Yaskawa INFORM job: R1_W29-KM-NOWY.JBI

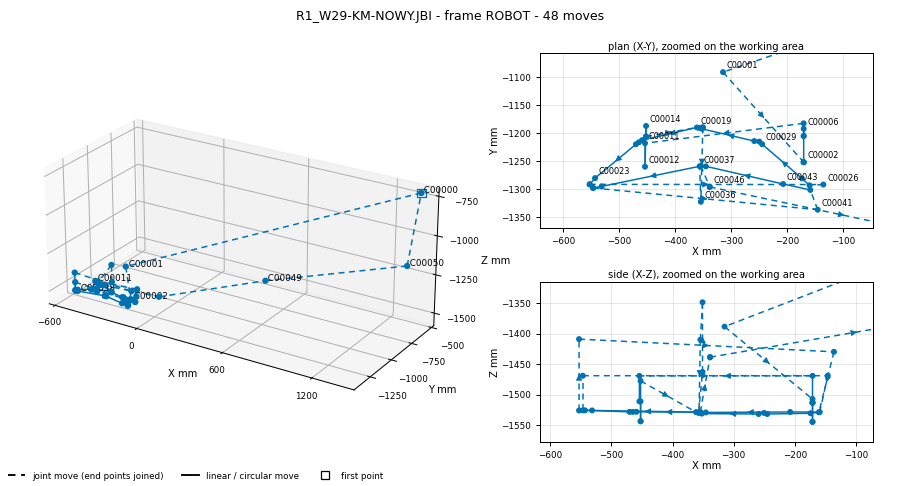
[picture p0: tool path of R1_W29-KM-NOWY.JBI in frame ROBOT, 48 of 48 moves have a stored position in this frame; points joined in program order, loops and branches not executed]
/JOB
//NAME R1_W29-KM-NOWY
///FOLDERNAME KRIS-SCIANA
//POS
///NPOS 52,52,48,3,0,0
///TOOL 0
///POSTYPE ROBOT
///RECTAN
///RCONF 0,0,0,0,0,0,0,0,0,0,0,0,0,0,0,0,0,0,0,0,0,0,0,0
C00000=1380.020,-512.213,-734.768,45.7984,-2.5734,-62.2106
C00001=-314.885,-1091.342,-1388.620,7.0991,47.6528,95.5247
C00002=-170.882,-1252.122,-1507.196,7.0965,47.6516,95.5184
C00003=-170.878,-1252.127,-1513.169,7.0965,47.6519,95.5192
C00004=-170.856,-1252.136,-1525.077,7.0962,47.6516,95.5223
C00005=-170.878,-1252.127,-1513.169,7.0965,47.6519,95.5192
C00006=-170.880,-1192.452,-1513.156,7.0958,47.6523,95.5184
C00007=-170.881,-1205.262,-1544.508,7.0940,47.6532,95.5150
C00008=-170.883,-1210.138,-1544.498,7.0940,47.6527,95.5159
C00009=-170.881,-1205.262,-1544.508,7.0940,47.6532,95.5150
C00010=-170.885,-1182.718,-1469.214,7.0949,47.6534,95.5162
C00011=-454.226,-1218.230,-1469.227,7.0938,47.6529,95.5164
C00012=-454.225,-1260.141,-1510.984,7.0936,47.6521,95.5169
C00013=-454.221,-1260.145,-1522.091,7.0917,47.6525,95.5139
C00014=-452.331,-1187.443,-1510.977,7.0932,47.6531,95.5154
C00015=-452.309,-1206.496,-1543.511,7.0905,47.6535,95.5128
C00016=-452.283,-1211.717,-1543.520,7.0889,47.6539,95.5119
C00017=-452.309,-1206.496,-1543.511,7.0905,47.6535,95.5128
C00018=-452.308,-1206.485,-1477.500,7.0906,47.6527,95.5130
C00019=-361.495,-1190.117,-1528.559,4.0105,46.8580,82.9369
C00020=-459.241,-1212.758,-1528.059,4.0090,46.8598,82.9290
C00021=-465.152,-1216.573,-1528.195,4.0138,46.8598,102.2526
C00022=-470.424,-1220.169,-1528.108,4.0135,46.8596,110.5818
C00023=-543.410,-1280.537,-1525.621,4.0159,46.8611,110.5850
C00024=-553.033,-1291.721,-1525.884,4.0182,46.8612,110.5866
C00025=-553.029,-1291.719,-1409.041,4.0170,46.8613,110.5846
C00026=-135.797,-1292.057,-1429.838,4.0180,46.8613,34.2800
C00027=-160.429,-1293.450,-1528.859,4.0112,46.8630,34.2695
C00028=-174.166,-1280.960,-1530.412,4.0163,46.8653,34.2766
C00029=-245.014,-1220.022,-1531.655,4.0137,46.8657,34.2760
C00030=-250.213,-1215.388,-1529.872,4.0121,46.8638,62.9323
C00031=-259.100,-1214.397,-1531.605,4.0118,46.8648,62.9324
C00032=-352.156,-1192.622,-1530.999,4.0138,46.8647,62.9360
C00033=-357.322,-1190.843,-1529.939,4.0131,46.8635,62.9345
C00034=-350.946,-1189.951,-1462.802,4.0124,46.8636,62.9333
C00035=-350.944,-1189.951,-1348.723,4.0127,46.8636,62.9343
C00036=-354.498,-1322.808,-1410.027,-15.4920,32.5646,-91.9565
C00037=-356.649,-1259.427,-1528.581,-15.4938,32.5644,-91.9586
C00038=-531.724,-1295.391,-1525.761,-15.4977,32.5637,-91.9664
C00039=-546.841,-1298.072,-1525.633,-15.4952,32.5617,-91.9642
C00040=-546.841,-1298.137,-1468.923,-15.4951,32.5627,-91.9631
C00041=-145.871,-1337.003,-1468.926,-15.4954,32.5637,-91.9623
C00042=-159.004,-1301.691,-1528.387,-15.4958,32.5640,-91.9617
C00043=-207.491,-1291.075,-1528.320,-15.4966,32.5644,-91.9616
C00044=-345.558,-1259.505,-1529.077,-15.4968,32.5617,-91.9666
C00045=-354.594,-1258.772,-1528.388,-15.4965,32.5625,-91.9640
C00046=-338.619,-1296.215,-1438.631,-18.1913,27.2183,-112.1098
C00047=-338.616,-1296.213,-1438.634,-18.1910,27.2179,-81.5660
C00048=133.748,-1396.204,-1357.645,-19.2328,23.1684,-62.3382
C00049=800.262,-1291.531,-1131.161,-1.6815,44.3835,75.7924
C00050=1382.830,-664.674,-1139.962,22.7477,31.6881,-179.3432
C00051=1380.020,-512.213,-734.768,45.7984,-2.5734,-62.2106
BC00000=786.429,2790.581,1999.643
BC00001=1673.587,2787.026,1999.675
BC00002=1673.587,2787.026,1999.675
BC00003=1673.587,2787.026,1999.675
BC00004=1673.587,2787.026,1999.675
BC00005=1673.587,2787.026,1999.675
BC00006=1673.587,2787.026,1999.675
BC00007=1673.587,2787.026,1999.675
BC00008=1673.587,2787.026,1999.675
BC00009=1673.587,2787.026,1999.675
BC00010=1673.587,2787.026,1999.675
BC00011=1673.587,2787.026,1999.675
BC00012=1673.587,2787.026,1999.675
BC00013=1673.587,2787.026,1999.675
BC00014=1673.587,2787.026,1999.675
BC00015=1673.587,2787.026,1999.675
BC00016=1673.587,2787.026,1999.675
BC00017=1673.587,2787.026,1999.675
BC00018=1673.587,2787.026,1999.675
BC00019=1724.246,2786.825,1999.677
BC00020=1724.246,2786.825,1999.677
BC00021=1724.246,2786.825,1999.677
BC00022=1724.246,2786.825,1999.677
BC00023=1724.246,2786.825,1999.677
BC00024=1724.246,2786.825,1999.677
BC00025=1724.246,2786.825,1999.677
BC00026=1724.246,2786.825,1999.677
BC00027=1724.246,2786.825,1999.677
BC00028=1724.246,2786.825,1999.677
BC00029=1724.246,2786.825,1999.677
BC00030=1724.246,2786.825,1999.677
BC00031=1724.246,2786.825,1999.677
BC00032=1724.246,2786.825,1999.677
BC00033=1724.246,2786.825,1999.677
BC00034=1724.246,2786.825,1999.677
BC00035=1724.246,2786.825,1999.677
BC00036=1724.246,2786.825,1999.677
BC00037=1724.246,2786.825,1999.677
BC00038=1724.246,2786.825,1999.677
BC00039=1724.246,2786.825,1999.677
BC00040=1724.246,2786.825,1999.677
BC00041=1724.246,2786.825,1999.677
BC00042=1724.246,2786.825,1999.677
BC00043=1724.246,2786.825,1999.677
BC00044=1724.246,2786.825,1999.677
BC00045=1724.246,2786.825,1999.677
BC00046=1724.246,2786.825,1999.677
BC00047=1724.246,2786.825,1999.677
BC00048=1442.256,2786.825,1999.677
BC00049=812.904,2786.825,1999.677
BC00050=213.733,2786.825,1999.677
BC00051=786.429,2790.581,1999.643
///POSTYPE PULSE
///PULSE
EC00000=798155,-556476
EC00001=798156,-556476
EC00002=798156,-556476
EC00003=798156,-556476
EC00004=798156,-556476
EC00005=798156,-556476
EC00006=798156,-556476
EC00007=798156,-556476
EC00008=798156,-556476
EC00009=798156,-556476
EC00010=798156,-556476
EC00011=798156,-556476
EC00012=798156,-556476
EC00013=798156,-556476
EC00014=798156,-556476
EC00015=798156,-556476
EC00016=798156,-556476
EC00017=798156,-556476
EC00018=798156,-556476
EC00019=798156,-556476
EC00020=798156,-556476
EC00021=798156,-556476
EC00022=798156,-556476
EC00023=798156,-556476
EC00024=798156,-556476
EC00025=798156,-556476
EC00026=798156,-556476
EC00027=798156,-556476
EC00028=798156,-556476
EC00029=798156,-556476
EC00030=798156,-556476
EC00031=798156,-556476
EC00032=798156,-556476
EC00033=798156,-556476
EC00034=798156,-556476
EC00035=798156,-556476
EC00036=798156,-556476
EC00037=798156,-556476
EC00038=798156,-556476
EC00039=798156,-556476
EC00040=798156,-556476
EC00041=798156,-556476
EC00042=798156,-556476
EC00043=798156,-556476
EC00044=798156,-556476
EC00045=798156,-556476
EC00046=798156,-556476
EC00047=798155,-556476
///POSTYPE BASE
///RECTAN
///RCONF 0,0,0,0,1,0,0,0,0,0,0,0,0,0,0,0,0,0,0,0,0,0,0,0
P00006=2.006,1.622,-0.565,0.0000,0.0000,0.0000
P00021=0.073,2.058,-0.109,0.0000,0.0000,0.0000
P00022=2.006,1.622,-0.565,0.0000,0.0000,0.0000
//INST
///DATE 2024/02/06 17:41
///ATTR SC,RW,RJ
////FRAME ROBOT
///GROUP1 RB1,BS1
///GROUP2 ST1
NOP
MOVJ C00000 BC00000 VJ=15.00  +MOVJ EC00000 VJ=15.00
MOVJ C00001 BC00001 VJ=50.00  +MOVJ EC00001 VJ=50.00
MOVJ C00002 BC00002 VJ=15.00  +MOVJ EC00002 VJ=15.00
MOVL C00003 BC00003 V=58.3  +MOVJ EC00003 VJ=15.00
REFP 3 RB1 C00004 BC00004
CALL JOB:SEARCH-R1
SET P021 P006
SFTON P021
MOVL C00005 BC00005 V=58.3  +MOVJ EC00004 VJ=15.00
MOVL C00006 BC00006 V=58.3  +MOVJ EC00005 VJ=15.00
MOVL C00007 BC00007 V=58.3  +MOVJ EC00006 VJ=15.00
REFP 3 RB1 C00008 BC00008
CALL JOB:SEARCH-R1
SET P021 P006
SFTON P021
MOVL C00009 BC00009 V=58.3  +MOVJ EC00007 VJ=15.00
SFTOF
MOVL C00010 BC00010 V=133.3  +MOVJ EC00008 VJ=15.00
MOVJ C00011 BC00011 VJ=15.00  +MOVJ EC00009 VJ=15.00
MOVL C00012 BC00012 V=58.3  +MOVJ EC00010 VJ=15.00
REFP 3 RB1 C00013 BC00013
CALL JOB:SEARCH-R1
SET P022 P006
SFTON P022
MOVL C00014 BC00014 V=58.3  +MOVJ EC00011 VJ=15.00
MOVL C00015 BC00015 V=58.3  +MOVJ EC00012 VJ=15.00
REFP 3 RB1 C00016 BC00016
CALL JOB:SEARCH-R1
SET P022 P006
SFTON P022
MOVL C00017 BC00017 V=58.3  +MOVJ EC00013 VJ=15.00
SFTOF
MOVL C00018 BC00018 V=133.3  +MOVJ EC00014 VJ=15.00
SFTON P022
MOVJ C00019 BC00019 VJ=15.00  +MOVJ EC00015 VJ=50.00
MACRO1 MJ#(0) ARGF7
ARCON
MOVL C00020 BC00020 V=10.8  +MOVJ EC00016 VJ=15.00
MOVL C00021 BC00021 V=10.8  +MOVJ EC00017 VJ=15.00
MOVL C00022 BC00022 V=10.8  +MOVJ EC00018 VJ=15.00
MOVL C00023 BC00023 V=10.8  +MOVJ EC00019 VJ=15.00
MOVL C00024 BC00024 V=10.8  +MOVJ EC00020 VJ=15.00
ARCOF
SFTOF
MOVJ C00025 BC00025 VJ=15.00  +MOVJ EC00021 VJ=15.00
MOVJ C00026 BC00026 VJ=15.00  +MOVJ EC00022 VJ=15.00
SFTON P021
MOVJ C00027 BC00027 VJ=15.00  +MOVJ EC00023 VJ=15.00
ARCON
MOVL C00028 BC00028 V=10.8  +MOVJ EC00024 VJ=15.00
MOVL C00029 BC00029 V=10.8  +MOVJ EC00025 VJ=15.00
MOVL C00030 BC00030 V=10.8  +MOVJ EC00026 VJ=15.00
MOVL C00031 BC00031 V=10.8  +MOVJ EC00027 VJ=15.00
MOVL C00032 BC00032 V=10.8  +MOVJ EC00028 VJ=15.00
MOVL C00033 BC00033 V=10.8  +MOVJ EC00029 VJ=15.00
ARCOF
MOVJ C00034 BC00034 VJ=15.00  +MOVJ EC00030 VJ=15.00
SFTOF
MOVJ C00035 BC00035 VJ=15.00  +MOVJ EC00031 VJ=15.00
MOVJ C00036 BC00036 VJ=15.00  +MOVJ EC00032 VJ=15.00
SFTON P022
MOVJ C00037 BC00037 VJ=15.00  +MOVJ EC00033 VJ=15.00
ARCON
MOVL C00038 BC00038 V=10.8  +MOVJ EC00034 VJ=15.00
MOVL C00039 BC00039 V=10.8  +MOVJ EC00035 VJ=15.00
ARCOF
MOVJ C00040 BC00040 VJ=15.00  +MOVJ EC00036 VJ=15.00
SFTOF
MOVJ C00041 BC00041 VJ=15.00  +MOVJ EC00037 VJ=15.00
SFTON P021
MOVJ C00042 BC00042 VJ=15.00  +MOVJ EC00038 VJ=15.00
ARCON
MOVL C00043 BC00043 V=10.8  +MOVJ EC00039 VJ=15.00
MOVL C00044 BC00044 V=10.8  +MOVJ EC00040 VJ=15.00
MOVL C00045 BC00045 V=10.8  +MOVJ EC00041 VJ=15.00
ARCOF
MOVJ C00046 BC00046 VJ=15.00  +MOVJ EC00042 VJ=15.00
MOVJ C00047 BC00047 VJ=20.00  +MOVJ EC00043 VJ=100.00
MOVJ C00048 BC00048 VJ=20.00  +MOVJ EC00044 VJ=20.00
SFTOF
MOVJ C00049 BC00049 VJ=20.00  +MOVJ EC00045 VJ=20.00
MOVJ C00050 BC00050 VJ=20.00  +MOVJ EC00046 VJ=20.00
MOVJ C00051 BC00051 VJ=100.00  +MOVJ EC00047 VJ=15.00
END
